FUNCTION_BLOCK FB_Stepper EXTENDS FB_StateMachine  IMPLEMENTS I_StateMachine
VAR_INPUT
	bStartHoming : BOOL;

END_VAR
VAR
	eInnerState : E_StepperStates;
	fbHoming	: FB_StepperHoming;
	stAxis		: ST_StepperAxis;
END_VAR

OuterLopSM();

PROPERTY Angle : LREAL
GET
Angle := stAxis.stAxisRef.NcToPlc.ActPos;
END_GET
END_PROPERTY

METHOD Disable : BOOL

VAR
	bChildBusy  : BOOL := FALSE;
END_VAR
fbHoming(bActive:=FALSE);



IF fbHoming.Busy THEN
	bChildBusy := TRUE;
ELSIF fbHoming.bError THEN
	bChildBusy := TRUE;
	{warning 'TODO: trigger e-stop'}
	//	Stack trace and bError switching are reserved for inner loop
	fbHoming.ErrorAck:=TRUE;
END_IF



IF bChildBusy THEN
	Disable := FALSE;
ELSE
	Disable := TRUE;
END_IF
END_METHOD

PROPERTY ForceHoming : BOOL
GET
ForceHoming := stAxis.bForceHoming;
END_GET
SET
stAxis.bForceHoming := ForceHoming;
END_SET
END_PROPERTY

PROPERTY Homed : BOOL
GET
IF bActive THEN
	Homed := NOT fbHoming.HomingNeeded;
ELSE
	Homed :=  TRUE;;
END_IF
END_GET
END_PROPERTY

METHOD InnerLoopSM : BOOL
// update all children FBs
fbHoming();

CASE CyclicInnerCase(TO_STRING(eInnerState)) OF
	E_StepperStates.Idle:
		IF bStartHoming THEN
			bStartHoming := FALSE;
			ChangeInnerState(E_StepperStates.Homing1);
		END_IF

	E_StepperStates.Homing1:
		IF fbHoming.Busy THEN
			// fbHoming should never be busy here 	
			sErrorDetails := 'fbHoming.Busy = TRUE';
			fbEventHandler(eNapID:=E_Event.UNABLE_TO_START_TASK,sMessage:=sErrorDetails);
			bError := TRUE;	
		ELSE
			IF fbHoming.bError THEN
				sErrorDetails := 'fbHoming.bReady=FALSE';
				fbEventHandler(eNapID:=E_Event.UNABLE_TO_START_TASK,sMessage:=sErrorDetails);
				bError := TRUE;
			ELSE
				fbHoming.bStart:=TRUE;
				ChangeInnerState(E_StepperStates.Homing2);
			END_IF
		END_IF
		
		
	E_StepperStates.Homing2:
		IF fbHoming.Busy THEN
			// Wait... fbStepper still busy 			
		ELSE
			IF fbHoming.bError THEN
				fbEventHandler(eNapID:=E_Event.TASK_FAILED,sTrace:=fbHoming.EventTrace);
				fbHoming.ErrorAck:=TRUE;
				bError := TRUE;
			ELSE
				IF Homed THEN
					fbEventHandler(eNapID:=E_Event.REQUEST_COMPLETED);
					ChangeInnerState(E_StepperStates.Idle);
				ELSE
					sErrorDetails := 'Homed=FALSE';
					fbEventHandler(eNapID:=E_Event.TASK_FAILED,sMessage:=sErrorDetails);
					bError := TRUE;
				END_IF
			END_IF
		END_IF
END_CASE
END_METHOD

METHOD PUBLIC ReadStatus : BOOL
stAxis.stAxisRef.ReadStatus();
{warning 'TODO: Add additional checks to FB_Steepper.ReadStatus()'}
END_METHOD

METHOD Reset : BOOL
// reset variables specific to this FB 

// Reactivate children FBs
fbHoming.Active:=TRUE;
END_METHOD

METHOD Setup : BOOL
eStateMachineSourceID := eStateSourceID;

IF eStateMachineSourceID = E_StateSourceID.L_Arm_StepperMotor THEN
	stAxis.bOutwardsForward	:= TRUE;
	stAxis.bOutwardsBackwards	:= FALSE;
	stAxis.bInwardsForward		:= FALSE;
	stAxis.bInwardsBackwards	:= TRUE;
	stAxis.fHomePosition		:= SystemConfig.fLEFT_STEPPER_HOME_POSITION;
ELSE // eStateMachineSourceID = E_StateSourceID.R_Arm_StepperMotor
	stAxis.bOutwardsForward	:= FALSE;
	stAxis.bOutwardsBackwards	:= TRUE;
	stAxis.bInwardsForward		:= TRUE;
	stAxis.bInwardsBackwards	:= FALSE;
	stAxis.fHomePosition		:= SystemConfig.fRIGHT_STEPPER_HOME_POSITION;
END_IF

fbHoming(eStateSourceID := THIS^.eStateMachineSourceID +  E_StepperID_Offset.StepperHoming,
					aErrorLog:=THIS^.aErrorLog,
					nErrorLogIndex:=THIS^.nErrorLogIndex,
					stParentsAxis:=THIS^.stAxis);
					
SetInnerEnumeration(nStateEnum:=THIS^.eInnerState);
END_METHOD

END_FUNCTION_BLOCK

(* stored: Version 1.1.0.1, ProductVersion 3.1.4024.12
   POU FB_Stepper: Id {70f60fc6-e7cd-4d28-b5de-2b239a406e43}, SpecialFunc None
   Folder Properties: Id {8978cbc0-270d-489b-90d2-49bd092d7602}
   Property Angle: Id {6a7eed59-1def-45bb-a1f6-b22de50f0d77}
   Get Get: Id {41816775-b8e3-4ead-85bb-3a0203449ba0}
   Method Disable: Id {cd457282-6054-4be8-8fe6-e00d6a2d0dfc}
   Property ForceHoming: Id {e90b8952-b364-4724-9c87-aa02d65a0d4b}
   Get Get: Id {b143f5c3-52bd-42fa-b7f9-c7a0b9e5053e}
   Set Set: Id {53bca0f8-9de6-44d8-8acb-7f475a3caf04}
   Property Homed: Id {2c688af8-592a-467f-b482-d9ba991c7c22}
   Get Get: Id {230bc8aa-0217-406b-a7e6-0232193e7d7a}
   Method InnerLoopSM: Id {ee4afb9f-5861-4e61-a530-082a879b7012}
   Method ReadStatus: Id {43ddb076-e090-43b0-b179-31afad3c41f5}
   Method Reset: Id {d54bc836-7075-4a56-8e55-ca9951410268}
   Method Setup: Id {5802140c-bf45-4cf3-9f73-9432ea27d7bb} *)
